// TIA Portal V19 export
TYPE "LEXCHANGETRAY_typeAxisSimpleControlCommands_2"
// stored: Access Published
   STRUCT
      refreshConfiguration : Bool;
      editConfiguration : Bool;
      saveConfiguration : Bool;
      enableAxis : Bool;
      resetAxis : Bool;
      home : Bool;
      halt : Bool;
      posAbsolute : Bool;
      posRelative : Bool;
      moveVelocity : Bool;
      jogForward : Bool;
      jogBackward : Bool;
      stop : Bool;
      readValues : Bool;
      enableTorque : Bool;
   END_STRUCT;
END_TYPE
